{attribute addProperty BoxType "EL5151-0021-0018"}
{attribute addProperty Id "StatusAT %I*Status_5507CB4B1621Counter_valueAT %I*UDINT32417Latch_valueAT %I*UDINT32418"}
{attribute addProperty CRC "87803933"}
{attribute addProperty SizeInBites "80"}
{attribute addProperty SizeInBytes "10"}
TYPE ENC_Status_053BC81D :
STRUCT
	{attribute addProperty Name "Status"}
	Status AT %I* : Status_5507CB4B;
	{attribute addProperty Name "Counter_value"}
	Counter_value AT %I* : UDINT;
	{attribute addProperty Name "Latch_value"}
	Latch_value AT %I* : UDINT;
END_STRUCT
END_TYPE

(* stored: Version 1.2.0.0, ProductVersion 3.1.4024.9
   DUT ENC_Status_053BC81D: Id {e01363a7-d710-4c0a-b5ed-70a9fbf38ebd} *)
